// TIA Portal V16 export
// export: Created 2021-07-03T21:22:43.5741923Z, ExportSetting WithDefaults, DisplayName Totally Integrated Automation Portal, DisplayVersion V16, DisplayName TIA Portal Version Control Interface, DisplayVersion V16, DisplayName TIA Portal Openness, DisplayVersion V16, DisplayName STEP 7 Professional, DisplayVersion V16, DisplayName STEP 7 Safety, DisplayVersion V16, DisplayName WinCC Professional, DisplayVersion V16
TYPE "118MK2_UPIF_Cmd"
// stored: IsFailsafeCompliant false
   STRUCT
      COMMAND_P { ExternalAccessible := 'False'; ExternalVisible := 'False'; ExternalWritable := 'False'} : Byte;   // Command Request - Machine Commands.
      CURRENT_ACTIVE_RECIPE_P { ExternalAccessible := 'False'; ExternalVisible := 'False'; ExternalWritable := 'False'} : Byte := BYTE#16#01;   // Indicates the active remote recipe (value 1-15)
      REC_EJEC_DELAY_TIME_P { ExternalAccessible := 'False'; ExternalVisible := 'False'; ExternalWritable := 'False'} : Byte;   // Recipe: Ejector delay time - Unsigned 8 bit integer value. Range 0 to 50ms
      REC_EJEC_ON_TIME_P { ExternalAccessible := 'False'; ExternalVisible := 'False'; ExternalWritable := 'False'} : Byte;   // Recipe: Ejector on time - Unsigned 8 bit integer value. Range 1 to 50ms
      REC_ALG_BLINT_TH_P { ExternalAccessible := 'False'; ExternalVisible := 'False'; ExternalWritable := 'False'} : Word;   // Recipe: Algorithm blue intensity threshold - Unsigned 16 bit integer value. Range 60 to 10000mV
      REC_ALG_BLRED_DISC_OFF_P { ExternalAccessible := 'False'; ExternalVisible := 'False'; ExternalWritable := 'False'} : Word;   // Recipe: Algorithm blue-red discrimination offset - Unsigned 16 bit integer value. Range 0 to 10000mV
      REC_ALG_BLRED_DISC_RAT_P { ExternalAccessible := 'False'; ExternalVisible := 'False'; ExternalWritable := 'False'} : Word;   // Recipe: Algorithm blue-red discrimination ratio - Unsigned 16 bit integer value. Range 1 to 1000 (is gradient of 0.01 to 10.00)
      REC_VIB_FEED_SP_P { ExternalAccessible := 'False'; ExternalVisible := 'False'; ExternalWritable := 'False'} : Byte;   // Recipe: Vibratory feeder set-point, Unsigned 8 bit integer value. Range 0 to 100%
      REC_AUTO_FEED_CNTRL_P { ExternalAccessible := 'False'; ExternalVisible := 'False'; ExternalWritable := 'False'} : Bool;   // Recipe: Automatic feeder control - OFF(0) – No closed loop control, ON(1) – Closed loop control
      REC_RESERVED0_P { ExternalAccessible := 'False'; ExternalVisible := 'False'; ExternalWritable := 'False'} : Bool;   // Recipe: Reserved - Spare
      REC_RESERVED1_P { ExternalAccessible := 'False'; ExternalVisible := 'False'; ExternalWritable := 'False'} : Bool;   // Recipe: Reserved - Spare
      REC_RESERVED2_P { ExternalAccessible := 'False'; ExternalVisible := 'False'; ExternalWritable := 'False'} : Bool;   // Recipe: Reserved - Spare
      REC_RESERVED3_P { ExternalAccessible := 'False'; ExternalVisible := 'False'; ExternalWritable := 'False'} : Bool;   // Recipe: Reserved - Spare
      REC_RESERVED4_P { ExternalAccessible := 'False'; ExternalVisible := 'False'; ExternalWritable := 'False'} : Bool;   // Recipe: Reserved - Spare
      REC_RESERVED5_P { ExternalAccessible := 'False'; ExternalVisible := 'False'; ExternalWritable := 'False'} : Bool;   // Recipe: Reserved - Spare
      REC_RESERVED6_P { ExternalAccessible := 'False'; ExternalVisible := 'False'; ExternalWritable := 'False'} : Bool;   // Recipe: Reserved - Spare
      REC_GATE_POSITION_P { ExternalAccessible := 'False'; ExternalVisible := 'False'; ExternalWritable := 'False'} : Byte;   // Recipe: Gate position - Range 0 to 5, ‘0’ - No auto gate control, ‘1’ – Move gate to position 1(-2 +1mm), ‘2’ – Move gate to position 2(-4+2mm), ‘3’ – Move gate to position 3(-8+4mm), ‘4’ – Move gate to position 4(-16+8mm), ‘5’ – Move gate to position 5(-32+16mm)
      SPARE0_P { ExternalAccessible := 'False'; ExternalVisible := 'False'; ExternalWritable := 'False'} : Byte;   // Spare
      SPARE1_P { ExternalAccessible := 'False'; ExternalVisible := 'False'; ExternalWritable := 'False'} : DWord;   // Spare
      SPARE2_P { ExternalAccessible := 'False'; ExternalVisible := 'False'; ExternalWritable := 'False'} : DWord;   // Spare
      SPARE3_P { ExternalAccessible := 'False'; ExternalVisible := 'False'; ExternalWritable := 'False'} : Byte;   // Spare
      HEARTBEAT_MPLC_CRIOCONT { ExternalAccessible := 'False'; ExternalVisible := 'False'; ExternalWritable := 'False'} : Byte;   // Communication Heartbeat between Machine PLC and cRIO Controller. This value received from PLC is returned in status message to the PLC.
      USER_NAME_P { ExternalAccessible := 'False'; ExternalVisible := 'False'; ExternalWritable := 'False'} : Array[0..7] of Byte;   // User name for authorisation/addition on cRIO controller security lookup table, 8-character string. This field will contain the old password only for a password update request.
      USER_PASSWORD_P { ExternalAccessible := 'False'; ExternalVisible := 'False'; ExternalWritable := 'False'} : Array[0..7] of Byte;   // User password for authorisation/addition on cRIO Controller security lookup table, 8-character string. This field will contain the new password only for a password update request.
      USER_ACCESS_LEVEL_P { ExternalAccessible := 'False'; ExternalVisible := 'False'; ExternalWritable := 'False'} : Byte;   // User access level for addition on cRIO Controller security lookup table.
      SEC_LOOKUPTABLE_PNTR_P { ExternalAccessible := 'False'; ExternalVisible := 'False'; ExternalWritable := 'False'} : Byte;   // Lookup user in security lookup table. Range: 1 to 40, 0 - Hidden administrator.
      REMOTE_DS_INLK_P { ExternalAccessible := 'False'; ExternalVisible := 'False'; ExternalWritable := 'False'} : Bool;   // Status of the D/S int. on either MachPLC-H/W or PlntPLC-S/W 0 - DS interlocked, 1 - DS interlock healthy.
      RESERVED0 { ExternalAccessible := 'False'; ExternalVisible := 'False'; ExternalWritable := 'False'} : Bool;   // Reserved - Spare
      RESERVED1 { ExternalAccessible := 'False'; ExternalVisible := 'False'; ExternalWritable := 'False'} : Bool;   // Reserved - Spare
      RESERVED2 { ExternalAccessible := 'False'; ExternalVisible := 'False'; ExternalWritable := 'False'} : Bool;   // Reserved - Spare
      RESERVED3 { ExternalAccessible := 'False'; ExternalVisible := 'False'; ExternalWritable := 'False'} : Bool;   // Reserved - Spare
      RESERVED4 { ExternalAccessible := 'False'; ExternalVisible := 'False'; ExternalWritable := 'False'} : Bool;   // Reserved - Spare
      RESERVED5 { ExternalAccessible := 'False'; ExternalVisible := 'False'; ExternalWritable := 'False'} : Bool;   // Reserved - Spare
      RESERVED6 { ExternalAccessible := 'False'; ExternalVisible := 'False'; ExternalWritable := 'False'} : Bool;   // Reserved - Spare
      SPARE4_P { ExternalAccessible := 'False'; ExternalVisible := 'False'; ExternalWritable := 'False'} : Byte;   // Spare
      RTC_CMD { ExternalAccessible := 'False'; ExternalVisible := 'False'; ExternalWritable := 'False'; S7_SetPoint := 'True'} : "RTC";
      "Ejector Feedback Override Disable" { ExternalAccessible := 'False'; ExternalVisible := 'False'; ExternalWritable := 'False'} : Bool;   // 'State of 'Override Checker Cycle Sequence' control on the OTI Alarm page (0=Enabled; 1=Disabled)
      "Checker Cycle Override Disable" { ExternalAccessible := 'False'; ExternalVisible := 'False'; ExternalWritable := 'False'} : Bool;   // State of 'Override Ejector Sense Feedback Alarms' control on the OTI Alarm page (0=Enabled; 1=Disabled)
      RESERVED_2 { ExternalAccessible := 'False'; ExternalVisible := 'False'; ExternalWritable := 'False'} : Bool;   // Spare
      RESERVED_3 { ExternalAccessible := 'False'; ExternalVisible := 'False'; ExternalWritable := 'False'} : Bool;   // Spare
      RESERVED_4 { ExternalAccessible := 'False'; ExternalVisible := 'False'; ExternalWritable := 'False'} : Bool;   // Spare
      RESERVED_5 { ExternalAccessible := 'False'; ExternalVisible := 'False'; ExternalWritable := 'False'} : Bool;   // Spare
      RESERVED_6 { ExternalAccessible := 'False'; ExternalVisible := 'False'; ExternalWritable := 'False'} : Bool;   // Spare
      RESERVED_7 { ExternalAccessible := 'False'; ExternalVisible := 'False'; ExternalWritable := 'False'} : Bool;   // Spare
      SPARE5 { ExternalAccessible := 'False'; ExternalVisible := 'False'; ExternalWritable := 'False'} : Byte;   // Spare
      SPARE5_P { ExternalAccessible := 'False'; ExternalVisible := 'False'; ExternalWritable := 'False'} : Word;   // Spare
      SPARE6_P { ExternalAccessible := 'False'; ExternalVisible := 'False'; ExternalWritable := 'False'} : DWord;   // Spare
      SPARE7_P { ExternalAccessible := 'False'; ExternalVisible := 'False'; ExternalWritable := 'False'} : DWord;   // Spare
      SPARE8_P { ExternalAccessible := 'False'; ExternalVisible := 'False'; ExternalWritable := 'False'} : DWord;   // Spare
      SPARE9_P { ExternalAccessible := 'False'; ExternalVisible := 'False'; ExternalWritable := 'False'} : DWord;   // Spare
   END_STRUCT;
END_TYPE
